{attribute addProperty BoxType "EP9224-0023-0016"}
{attribute addProperty Id "Error_UsAT %I*BOOL811Error_UpAT %I*BOOL812Warning_UsAT %I*BOOL813Warning_UpAT %I*BOOL814Status_UsAT %I*BOOL815Status_UpAT %I*BOOL816Channel_ErrorAT %I*BOOL817Error_Sum_CurrentAT %I*BOOL818Warning_Sum_CurrentAT %I*BOOL819TxPDO_StateAT %I*BOOL8115TxPDO_ToggleAT %I*BOOL8116Current_UsAT %I*INT16217Current_UpAT %I*INT16218"}
{attribute addProperty CRC "1020903075"}
{attribute addProperty SizeInBites "120"}
{attribute addProperty SizeInBytes "15"}
TYPE DPO_Inputs_Channel_3CD9BEA3 :
STRUCT
	{attribute addProperty Name "Error_Us"}
	Error_Us AT %I* : BOOL;
	{attribute addProperty Name "Error_Up"}
	Error_Up AT %I* : BOOL;
	{attribute addProperty Name "Warning_Us"}
	Warning_Us AT %I* : BOOL;
	{attribute addProperty Name "Warning_Up"}
	Warning_Up AT %I* : BOOL;
	{attribute addProperty Name "Status_Us"}
	Status_Us AT %I* : BOOL;
	{attribute addProperty Name "Status_Up"}
	Status_Up AT %I* : BOOL;
	{attribute addProperty Name "Channel_Error"}
	Channel_Error AT %I* : BOOL;
	{attribute addProperty Name "Error_Sum_Current"}
	Error_Sum_Current AT %I* : BOOL;
	{attribute addProperty Name "Warning_Sum_Current"}
	Warning_Sum_Current AT %I* : BOOL;
	{attribute addProperty Name "TxPDO_State"}
	TxPDO_State AT %I* : BOOL;
	{attribute addProperty Name "TxPDO_Toggle"}
	TxPDO_Toggle AT %I* : BOOL;
	{attribute addProperty Name "Current_Us"}
	Current_Us AT %I* : INT;
	{attribute addProperty Name "Current_Up"}
	Current_Up AT %I* : INT;
END_STRUCT
END_TYPE

(* stored: Version 1.2.0.0, ProductVersion 3.1.4024.9
   DUT DPO_Inputs_Channel_3CD9BEA3: Id {1d2ce99d-8ff0-4141-a3cc-77ca63cd4298} *)
